// TIA Portal V20 export
DATA_BLOCK "GLOBAL_ROBOT_HMI_IF_DB"   // DB215
{ S7_Optimized_Access := 'TRUE' }
// stored: AutoNumber false, MemoryReserve 100
   VAR RETAIN
      Robot : Array[0..19] of "ROBOT_INTERFACE_HMI_UDT";
      Robot_HS { S7_SetPoint := 'True'} : Array[0..19] of "HS_HISTORY_HMI_UDT";
   END_VAR
BEGIN
   // Robot[1] : +ST020-RB01
   // Robot[2] : +ST020-RB02
   // Robot[3] : +ST020-RB03
   // Robot[4] : +ST020-RB04
   // Robot[5] : +ST020-RB06
   // Robot[6] : +ST025-RB01
   // Robot[7] : +ST025-RB02
   // Robot[8] : +ST030-RB01
   // Robot[9] : +ST030-RB02
   // Robot[10] : +ST030-RB03
   // Robot[11] : +ST030-RB04
END_DATA_BLOCK
